{attribute 'Tc2GvlVarNames'}
VAR_CONFIG
END_VAR

(* stored: Version 1.1.0.1, ProductVersion 3.1.4022.10
   GVL Variablen_Konfiguration: Id {d392f725-00ce-4b53-8297-c7cc32d4041b} *)
